TYPE ST_LastBatch :
STRUCT
	iType					:INT;
	sBatchNumber			:STRING;
	sRecipe					:STRING;
	sUser					:STRING;
	sStarted				:STRING;
	sFinished				:STRING;

END_STRUCT
END_TYPE

(* stored: Version 1.1.0.1, ProductVersion 3.1.4024.12
   DUT ST_LastBatch: Id {4890c9f9-f1b4-4fb4-912c-49e657486ee3} *)
